SUBAPPLICATION Uebung_039b_AX (* Spiegelabfolge V2 mit Schrittkette *)
  (* Standard: 61499-2; Description: Copyright (c) 2023 Meisterschulen am Ostbahnhof This program and the accompanying materials are made available under the terms of the Eclipse Public License 2.0 which is available at https://www.eclipse.org/legal/epl-2.0/ SPDX-License-Identifier: EPL-2.0 *)
  (* Version 1.0, 2023-10-23, Franz Höpfinger, Meisterschulen am Ostbahnhof, initial API and implementation and/or initial documentation *)
  PACKAGE Uebungen;
  IMPORT Uebungen::const::UT::DefaultPool::SoftKey_F1;
  IMPORT logiBUS::io::DQ::logiBUS_DO::Output_Q1;
  IMPORT logiBUS::io::DQ::logiBUS_DO::Output_Q2;
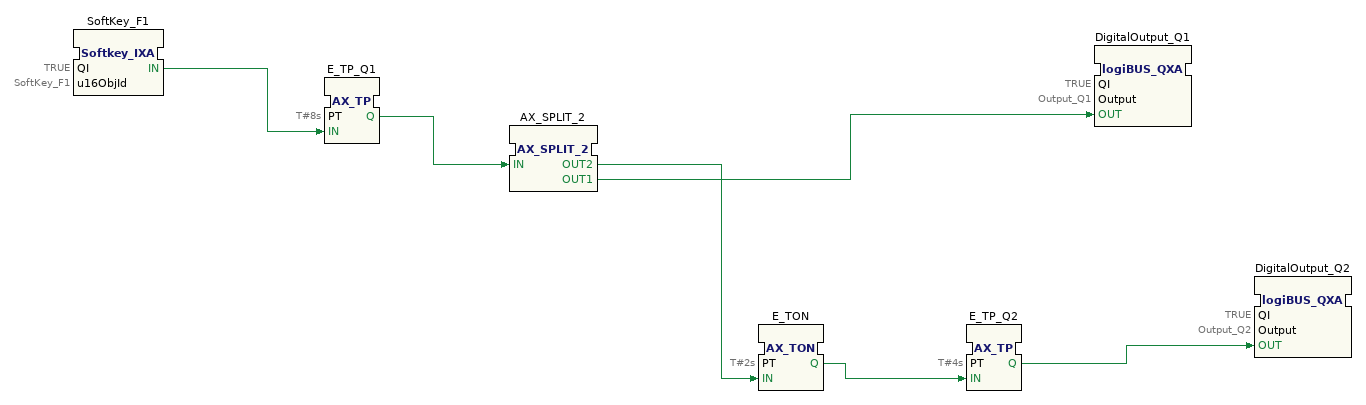
  FBS
    DigitalOutput_Q1 : logiBUS::io::DQ::logiBUS_QXA(QI := TRUE, Output := Output_Q1);
    DigitalOutput_Q2 : logiBUS::io::DQ::logiBUS_QXA(QI := TRUE, Output := Output_Q2);
    SoftKey_F1 : isobus::UT::io::Softkey::Softkey_IXA(QI := TRUE, u16ObjId := SoftKey_F1);
    E_TP_Q1 : adapter::events::unidirectional::timers::AX_TP(PT := T#8s);
    E_TP_Q2 : adapter::events::unidirectional::timers::AX_TP(PT := T#4s);
    E_TON : adapter::events::unidirectional::timers::AX_TON(PT := T#2s);
    AX_SPLIT_2 : adapter::events::unidirectional::AX_SPLIT_2;
  END_FBS
  ADAPTER_CONNECTIONS
    SoftKey_F1.IN TO E_TP_Q1.IN;
    E_TON.Q TO E_TP_Q2.IN;
    AX_SPLIT_2.OUT2 TO E_TON.IN;
    AX_SPLIT_2.OUT1 TO DigitalOutput_Q1.OUT;
    E_TP_Q2.Q TO DigitalOutput_Q2.OUT;
    E_TP_Q1.Q TO AX_SPLIT_2.IN;
  END_CONNECTIONS
END_SUBAPPLICATION
